# B&R Automation Studio project prac3
Automation Studio 4.5.2.102; technology packages: Acp10Arnc0 5.2.1

## Configuration Config1

CPU 4PP065.0571-P74, AutomationRuntime D4.52, Build 4.1.2, Vc V4.52.0, Safety 1.6

### Task classes (Cpu.sw)
```
Cyclic#1 (cycle 2000 us, tolerance 0 us):
  ncsdcctrl <- ncsdcctrl.prg
Cyclic#4:
  Program <- Program.prg
NcDataObjects: acp10etxen <- acp10etxen.dob, gAxis01a <- gAxis01obj.gAxis01a.dob, gAxis01i <- gAxis01obj.gAxis01i.dob, gAxis02a <- gAxis02obj.gAxis02a.dob, gAxis02i <- gAxis02obj.gAxis02i.dob, gAxis03a <- gAxis03obj.gAxis03a.dob, gAxis03i <- gAxis03obj.gAxis03i.dob, gAxis04a <- gAxis04obj.gAxis04a.dob, gAxis04i <- gAxis04obj.gAxis04i.dob
VcDataObjects: Visu <- Visu.dob
Libraries: Acp10man, Acp10par, NcGlobal, Acp10sdc, Acp10_MC, brsystem, sys_lib, runtime, AsBrStr, Library
```

### Hardware
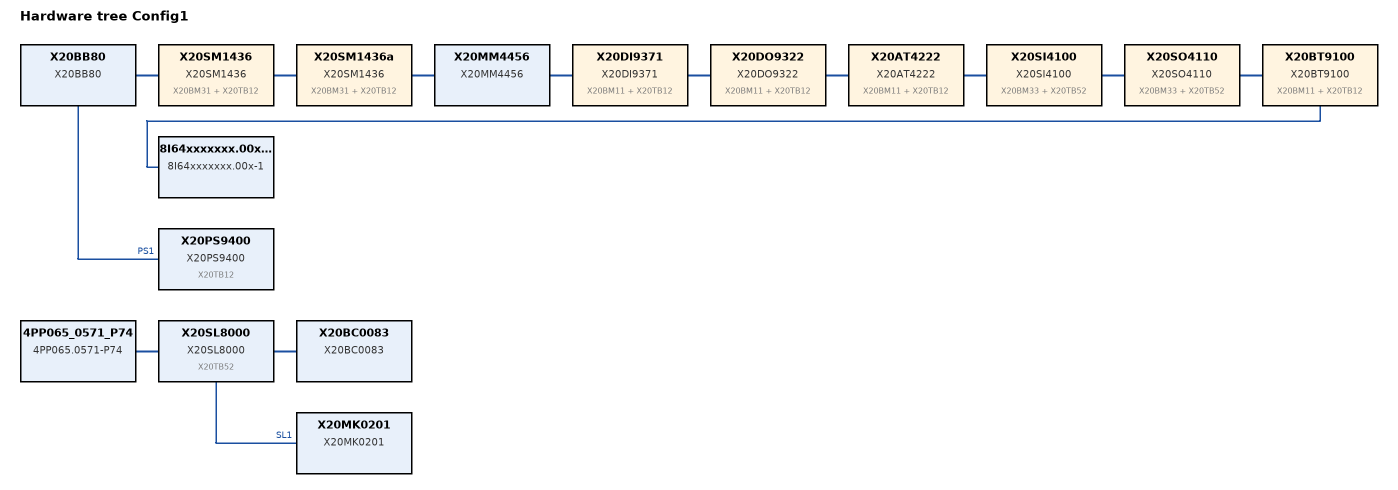
```
4PP065_0571_P74 : 4PP065.0571-P74 v1.1.2.0
  Connector IF5:
    ActivateDevice = 1
    Mode = Manual
    InternetAddress = 10.0.1.7
    SubnetMask = 255.255.255.0
  ConfigurationID = labBR
  TimerDeviceType = EPLX2X
  TimerDevice = 4PP065_0571_P74.IF4
  TaskClassIdleTime = 2000
  Cyclic1Duration = 2000
  Cyclic1Tolerance = 0
  Cyclic1Output = 1
  VcObjectName = Visu
8I64xxxxxxx.00x-1 : 8I64xxxxxxx.00x-1 v1.3.9.1  [X2X1 -> X20BT9100.X2X1 [Cable Type=X2XCable, Length=10, Version=1.0.0.2]]
  packedETAD = packed
  packedCMDD = packed
X20AT4222 : X20AT4222 v1.2.3.0  [SS1 -> X20TB12e.SS; SL -> X20BM11b.SL1]
X20BB80 : X20BB80 v1.0.2.0
X20BC0083 : X20BC0083 v2.9.0.0  [PLK1 -> X20SL8000.PLK2 [Cable Type=PowerlinkCable, Length=10, Version=1.0.0.2]; SL -> X20BB80.SL1]
X20BM11 : X20BM11 v1.0.0.1  [X2X1 -> X20MM4456.X2X2]
X20BM11a : X20BM11 v1.0.0.1  [X2X1 -> X20BM11.X2X2]
X20BM11b : X20BM11 v1.0.0.1  [X2X1 -> X20BM11a.X2X2]
X20BM11c : X20BM11 v1.0.0.1  [X2X1 -> X20BM33a.X2X2]
X20BM31 : X20BM31 v1.0.0.1  [X2X1 -> X20BB80.IF1]
X20BM31a : X20BM31 v1.0.0.1  [X2X1 -> X20BM31.X2X2]
X20BM33 : X20BM33 v1.0.0.4  [X2X1 -> X20BM11b.X2X2]
X20BM33a : X20BM33 v1.0.0.4  [X2X1 -> X20BM33.X2X2]
X20BT9100 : X20BT9100 v1.0.3.0  [SS1 -> X20TB12f.SS; SL -> X20BM11c.SL1]
X20DI9371 : X20DI9371 v1.0.2.0  [SS1 -> X20TB12c.SS; SL -> X20BM11.SL1]
X20DO9322 : X20DO9322 v1.0.3.0  [SS1 -> X20TB12d.SS; SL -> X20BM11a.SL1]
X20MK0201 : X20MK0201 v1.0.0.0  [SL -> X20SL8000.SL1]
X20MM4456 : X20MM4456 v1.4.0.0  [X2X1 -> X20BM31a.X2X2]
X20PS9400 : X20PS9400 v1.0.2.4  [SS1 -> X20TB12.SS; PS -> X20BB80.PS1]
X20SI4100 : X20SI4100 v1.10.1.1  [SS1 -> X20TB52a.SS; SL -> X20BM33.SL1]
X20SL8000 : X20SL8000 v1.6.5.1  [PLK1 -> 4PP065_0571_P74.IF4 [Cable Type=PowerlinkCable, Length=10, Version=1.0.0.2]; PLK2 -> X20BC0083.PLK1 [Cable Type=PowerlinkCable, Length=10, Version=1.0.0.2]; SS1 -> X20TB52.SS]
  SafeProject = SafeLOGIC-1
X20SM1436 : X20SM1436 v1.4.2.1  [SS1 -> X20TB12b.SS; SL -> X20BM31.SL1]
X20SM1436a : X20SM1436 v1.4.2.1  [SS1 -> X20TB12a.SS; SL -> X20BM31a.SL1]
X20SO4110 : X20SO4110 v1.10.1.1  [SS1 -> X20TB52b.SS; SL -> X20BM33a.SL1]
  SafeModuleID = 3
X20TB12 : X20TB12 v1.0.0.0
X20TB12a : X20TB12 v1.0.0.0
X20TB12b : X20TB12 v1.0.0.0
X20TB12c : X20TB12 v1.0.0.0
X20TB12d : X20TB12 v1.0.0.0
X20TB12e : X20TB12 v1.0.0.0
X20TB12f : X20TB12 v1.0.0.0
X20TB52 : X20TB52 v1.0.0.1
X20TB52a : X20TB52 v1.0.0.1
X20TB52b : X20TB52 v1.0.0.1
```

### IoMap.iom - 4PP065_0571_P74/IoMap.iom
```iecst
VAR_CONFIG
	Cyclic#1.gAxis01_DrvIf.iLifeCnt AT %IB."X20SM1436".LifeCnt;
	Cyclic#1.gAxis01_DrvIf.iDrvOK AT %IX."X20SM1436".DrvOk01;
	Cyclic#1.gAxis01_DrvIf.oBoostCurrent AT %QX."X20SM1436".BoostCurrent01;
	Cyclic#1.gAxis01_DrvIf.oStandStillCurrent AT %QX."X20SM1436".StandstillCurrent01;
	Cyclic#1.gAxis01_DrvIf.oSetTime AT %QW."X20SM1436".SetTime01;
	Cyclic#1.gAxis01_MotorStep0 AT %QW."X20SM1436".Motor1Step0;
	Cyclic#1.gAxis01_DiDoIf.iLifeCntDriveEnable AT %IB."X20SM1436".LifeCnt;
	Cyclic#1.gAxis01_DiDoIf.iLifeCntDriveReady AT %IB."X20SM1436".LifeCnt;
	Cyclic#1.gAxis01_DiDoIf.iDriveReady AT %IX."X20SM1436".DrvOk01;
	Cyclic#1.gAxis01_DiDoIf.oDriveEnable AT %QX."X20SM1436".DriveEnable01;
	Cyclic#1.gAxis01_EncIf1.iLifeCnt AT %IB."X20SM1436".LifeCnt;
	Cyclic#1.gAxis01_EncIf1.iEncOK AT %IX."X20SM1436".EncOk01;
	Cyclic#1.gAxis01_EncIf1.iActPos AT %IW."X20SM1436".ActPos01;
	Cyclic#1.gAxis01_EncIf1.iRefPulsePos AT %IW."X20SM1436".RefPulsePos01;
	Cyclic#1.gAxis01_EncIf1.iRefPulseCnt AT %IB."X20SM1436".RefPulseCnt01;
	Cyclic#1.gAxis01_EncIf1.iActTime AT %IW."X20SM1436".ActTime01;
	Cyclic#1.gAxis02_DrvIf.iLifeCnt AT %IB."X20SM1436a".LifeCnt;
	Cyclic#1.gAxis02_DrvIf.iDrvOK AT %IX."X20SM1436a".DrvOk01;
	Cyclic#1.gAxis02_DrvIf.oBoostCurrent AT %QX."X20SM1436a".BoostCurrent01;
	Cyclic#1.gAxis02_DrvIf.oStandStillCurrent AT %QX."X20SM1436a".StandstillCurrent01;
	Cyclic#1.gAxis02_DrvIf.oSetTime AT %QW."X20SM1436a".SetTime01;
	Cyclic#1.gAxis02_MotorStep0 AT %QW."X20SM1436a".Motor1Step0;
	Cyclic#1.gAxis02_DiDoIf.iLifeCntDriveEnable AT %IB."X20SM1436a".LifeCnt;
	Cyclic#1.gAxis02_DiDoIf.iLifeCntDriveReady AT %IB."X20SM1436a".LifeCnt;
	Cyclic#1.gAxis02_DiDoIf.iDriveReady AT %IX."X20SM1436a".DrvOk01;
	Cyclic#1.gAxis02_DiDoIf.oDriveEnable AT %QX."X20SM1436a".DriveEnable01;
	Cyclic#1.gAxis02_EncIf1.iLifeCnt AT %IB."X20SM1436a".LifeCnt;
	Cyclic#1.gAxis02_EncIf1.iEncOK AT %IX."X20SM1436a".EncOk01;
	Cyclic#1.gAxis02_EncIf1.iActPos AT %IW."X20SM1436a".ActPos01;
	Cyclic#1.gAxis02_EncIf1.iRefPulsePos AT %IW."X20SM1436a".RefPulsePos01;
	Cyclic#1.gAxis02_EncIf1.iRefPulseCnt AT %IB."X20SM1436a".RefPulseCnt01;
	Cyclic#1.gAxis02_EncIf1.iActTime AT %IW."X20SM1436a".ActTime01;
	Cyclic#1.gAxis04_DrvIf.iLifeCnt AT %IB."8I64xxxxxxx.00x-1".SDC_LifeCnt;
	Cyclic#1.gAxis04_DrvIf.iDrvOK AT %IX."8I64xxxxxxx.00x-1".ETAD_Input_Bool_02;
	Cyclic#1.gAxis04_DrvIf.oSetTime AT %QW."8I64xxxxxxx.00x-1".SDC_SetTime;
	Cyclic#1.::Program:speed AT %QW."8I64xxxxxxx.00x-1".LFRD_Output;
	Cyclic#1.gAxis04_DiDoIf.iLifeCntDriveReady AT %IB."8I64xxxxxxx.00x-1".SDC_LifeCnt;
	Cyclic#1.gAxis04_DiDoIf.iLifeCntDriveEnable AT %IB."8I64xxxxxxx.00x-1".SDC_LifeCnt;
	Cyclic#1.gAxis04_DiDoIf.oDriveEnable AT %QX."8I64xxxxxxx.00x-1".CMDD_Output_Bool_00;
	Cyclic#1.gAxis04_ModuleOk AT %QX."8I64xxxxxxx.00x-1".CMDD_Output_Bool_01;
	Cyclic#1.gAxis04_ModuleOk AT %QX."8I64xxxxxxx.00x-1".CMDD_Output_Bool_02;
	Cyclic#1.gAxis04_ModuleOk AT %IX."8I64xxxxxxx.00x-1".ModuleOk;
	Cyclic#1.gAxis04_DiDoIf.oDriveEnable AT %QX."8I64xxxxxxx.00x-1".CMDD_Output_Bool_03;
	Cyclic#1.gAxis04_DiDoIf.iDriveReady AT %IX."8I64xxxxxxx.00x-1".ETAD_Input_Bool_02;
	::Program:DRIVE.STATE AT %IW."8I64xxxxxxx.00x-1".ETAD_Input;
	::Program:DRIVE.COM AT %QW."8I64xxxxxxx.00x-1".CMDD_Output;
END_VAR
```

### Acp10map.ncm - 4PP065_0571_P74/Motion/Acp10map.ncm
```
NcMapping (NcSwId=Acp10)
  NcObject gAxis01 (ModuleId=X20SM1436, ModuleAddress=SDC_IF1.ST1, Type=ncAXIS, Channel=1, AcoposSimulation=Off, InitParameter=gAxis01i, AcoposParameter=gAxis01a, Disabled=FALSE, ModuleDisabled=FALSE)
  NcObject gAxis02 (ModuleId=X20SM1436a, ModuleAddress=SDC_IF1.ST2, Type=ncAXIS, Channel=1, AcoposSimulation=Off, InitParameter=gAxis02i, AcoposParameter=gAxis02a, Disabled=FALSE, ModuleDisabled=FALSE)
  NcObject gAxis04 (ModuleId=8I64xxxxxxx.00x-1, ModuleAddress=SDC_IF1.ST3, Type=ncAXIS, Channel=1, AcoposSimulation=Off, InitParameter=gAxis04i, AcoposParameter=gAxis04a, Disabled=FALSE, ModuleDisabled=FALSE)
```

## Logical view

Binary libraries used (declarations not repeated): operator, runtime, astime, AsIecCon, Acp10man, Acp10par, NcGlobal, Acp10sdc, Acp10_MC, brsystem, sys_lib, AsBrStr

### Global.var - Global variables
```iecst
VAR
	gAxis01 : ACP10AXIS_typ;
	gAxis01_HW : SdcHwCfg_typ := (0);
	gAxis01_DrvIf : SdcDrvIf16_typ := (0);
	gAxis01_EncIf1 : SdcEncIf16_typ := (0);
	gAxis01_DiDoIf : SdcDiDoIf_typ := (0);
	gAxis01_MotorStep0 : INT := (0);
	gAxis02 : ACP10AXIS_typ;
	gAxis02_HW : SdcHwCfg_typ := (0);
	gAxis02_DrvIf : SdcDrvIf16_typ := (0);
	gAxis02_EncIf1 : SdcEncIf16_typ := (0);
	gAxis02_DiDoIf : SdcDiDoIf_typ := (0);
	gAxis02_MotorStep0 : INT := (0);
	gAxis03 : ACP10AXIS_typ;
	gAxis03_HW : SdcHwCfg_typ := (0);
	gAxis03_DrvIf : SdcDrvIf16_typ := (0);
	gAxis03_DiDoIf : SdcDiDoIf_typ := (0);
	gAxis03_ModuleOk : BOOL := 0;
	gAxis04 : ACP10AXIS_typ;
	gAxis04_HW : SdcHwCfg_typ := (0);
	gAxis04_DrvIf : SdcDrvIf16_typ := (0);
	gAxis04_DiDoIf : SdcDiDoIf_typ := (0);
	gAxis04_ModuleOk : BOOL := 0;
	ENABLED : BOOL := FALSE;
END_VAR
```

### Package Logical/Libraries - Global libraries

### Library Logical/Libraries/Library (ANSIC)

#### Constants.var - Exported constants
```iecst
VAR CONSTANT
	CMD_SWITCHED_ON : UINT := 7;
	CMD_DISABLE_VOLTAGE1 : UINT := 0;
	CMD_ENABLED : UINT := 15;
	CMD_SHUTDOWN : UINT := 6;
	STATE_READY : UINT := 33;
	STATE_DISABLED : UINT := 64;
	STATE_SWITCHED_ON : UINT := 35;
END_VAR
```

#### Library.fun - Exported functions and function blocks
```iecst
{REDUND_OK} FUNCTION_BLOCK drive (*TODO: Add your comment here*) (*$GROUP=User,$CAT=User,$GROUPICON=User.png,$CATICON=User.png*)
	VAR_INPUT
		ENABLE : BOOL;
		STATE : UINT;
	END_VAR
	VAR_OUTPUT
		COM : UINT;
	END_VAR
END_FUNCTION_BLOCK
```

#### drive.c
```c
#include <bur/plctypes.h>
#ifdef __cplusplus
	extern "C"
	{
#endif
	#include "Library.h"
#ifdef __cplusplus
	};
#endif
/* TODO: Add your comment here */
void drive(struct drive* inst)
{
	UINT mask=inst->STATE & 0x6f;
	if(!inst->ENABLE){
		inst->COM = CMD_SHUTDOWN;
	}
	else{
		switch(mask)
		{
			case STATE_DISABLED:
				inst->COM=CMD_SHUTDOWN;
				break;
			case STATE_READY:
				inst->COM=CMD_ENABLED;
				break;
			case STATE_SWITCHED_ON:
				inst->COM=CMD_SWITCHED_ON;
				break;

		}
	}
}
```

### Program Logical/ncsdcctrl (IEC)

#### ncsdcctrl.var
```iecst
VAR
	gAxis01_oSetPosOld : INT := 0;
	gAxis02_oSetPosOld : INT := 0;
END_VAR
```

#### ncsdcctrlCyclic.st
```iecst
PROGRAM _CYCLIC

(* ### BEGIN gAxis01 ### *)

(* life counter emulation of digital inputs *)
      gAxis01_DiDoIf.iLifeCntReference := gAxis01_DiDoIf.iLifeCntReference + 1;
      gAxis01_DiDoIf.iLifeCntNegHwEnd  := gAxis01_DiDoIf.iLifeCntNegHwEnd  + 1;
      gAxis01_DiDoIf.iLifeCntPosHwEnd  := gAxis01_DiDoIf.iLifeCntPosHwEnd  + 1;

(* default function model of ACOPOSmicro: convert absolute steps to delta steps - overflow save delta calculation *)
      gAxis01_MotorStep0 := gAxis01_DrvIf.oSetPos - gAxis01_oSetPosOld;
      gAxis01_oSetPosOld := gAxis01_DrvIf.oSetPos;

(* ### END gAxis01 ### *)

(* ### BEGIN gAxis02 ### *)

(* life counter emulation of digital inputs *)
      gAxis02_DiDoIf.iLifeCntReference := gAxis02_DiDoIf.iLifeCntReference + 1;
      gAxis02_DiDoIf.iLifeCntNegHwEnd  := gAxis02_DiDoIf.iLifeCntNegHwEnd  + 1;
      gAxis02_DiDoIf.iLifeCntPosHwEnd  := gAxis02_DiDoIf.iLifeCntPosHwEnd  + 1;

(* default function model of ACOPOSmicro: convert absolute steps to delta steps - overflow save delta calculation *)
      gAxis02_MotorStep0 := gAxis02_DrvIf.oSetPos - gAxis02_oSetPosOld;
      gAxis02_oSetPosOld := gAxis02_DrvIf.oSetPos;

(* ### END gAxis02 ### *)

(* ### BEGIN gAxis03 ### *)

(* life counter emulation of digital inputs *)
        gAxis03_DiDoIf.iLifeCntReference := gAxis03_DiDoIf.iLifeCntReference + 1;
        gAxis03_DiDoIf.iLifeCntNegHwEnd  := gAxis03_DiDoIf.iLifeCntNegHwEnd  + 1;
        gAxis03_DiDoIf.iLifeCntPosHwEnd  := gAxis03_DiDoIf.iLifeCntPosHwEnd  + 1;

(* ### END gAxis03 ### *)

(* ### BEGIN gAxis04 ### *)

(* life counter emulation of digital inputs *)
        gAxis04_DiDoIf.iLifeCntReference := gAxis04_DiDoIf.iLifeCntReference + 1;
        gAxis04_DiDoIf.iLifeCntNegHwEnd  := gAxis04_DiDoIf.iLifeCntNegHwEnd  + 1;
        gAxis04_DiDoIf.iLifeCntPosHwEnd  := gAxis04_DiDoIf.iLifeCntPosHwEnd  + 1;

(* ### END gAxis04 ### *)

END_PROGRAM
```

#### ncsdcctrlInit.st
```iecst
PROGRAM _INIT

(* ### BEGIN gAxis01 ### *)

(* initialize general interfaces *)
      gAxis01.size := gAxis01.size;
      gAxis01_HW.DrvIf_Typ := ncSDC_DRVSM16;
      brsstrcpy( ADR(gAxis01_HW.DrvIf_Name[0]), ADR('gAxis01_DrvIf') );
      gAxis01_HW.DiDoIf_Typ := ncSDC_DIDO;
      brsstrcpy( ADR(gAxis01_HW.DiDoIf_Name[0]), ADR('gAxis01_DiDoIf') );
      gAxis01_HW.EncIf1_Typ := ncSDC_ENC16;
      brsstrcpy( ADR(gAxis01_HW.EncIf1_Name[0]), ADR('gAxis01_EncIf1') );
      gAxis01_EncIf1.iLifeCnt := gAxis01_EncIf1.iLifeCnt;

(* initialize old-value for delta step calculation *)
      gAxis01_oSetPosOld := gAxis01_DrvIf.oSetPos;

(* ### END gAxis01 ### *)

(* ### BEGIN gAxis02 ### *)

(* initialize general interfaces *)
      gAxis02.size := gAxis02.size;
      gAxis02_HW.DrvIf_Typ := ncSDC_DRVSM16;
      brsstrcpy( ADR(gAxis02_HW.DrvIf_Name[0]), ADR('gAxis02_DrvIf') );
      gAxis02_HW.DiDoIf_Typ := ncSDC_DIDO;
      brsstrcpy( ADR(gAxis02_HW.DiDoIf_Name[0]), ADR('gAxis02_DiDoIf') );
      gAxis02_HW.EncIf1_Typ := ncSDC_ENC16;
      brsstrcpy( ADR(gAxis02_HW.EncIf1_Name[0]), ADR('gAxis02_EncIf1') );
      gAxis02_EncIf1.iLifeCnt := gAxis02_EncIf1.iLifeCnt;

(* initialize old-value for delta step calculation *)
      gAxis02_oSetPosOld := gAxis02_DrvIf.oSetPos;

(* ### END gAxis02 ### *)

(* ### BEGIN gAxis03 ### *)

(* initialize variables *)
        gAxis03_HW.DrvIf_Typ := ncSDC_DRVSERVO16;
        brsstrcpy(ADR(gAxis03_HW.DrvIf_Name[0]), ADR('gAxis03_DrvIf'));
        gAxis03_HW.DiDoIf_Typ := ncSDC_DIDO;
        brsstrcpy(ADR(gAxis03_HW.DiDoIf_Name[0]), ADR('gAxis03_DiDoIf'));

(* force variable offset generation *)
        gAxis03.size                      := gAxis03.size;
        gAxis03_DrvIf.iLifeCnt            := gAxis03_DrvIf.iLifeCnt;
        gAxis03_DiDoIf.iLifeCntDriveReady := gAxis03_DiDoIf.iLifeCntDriveReady;
        gAxis03_ModuleOk                  := gAxis03_ModuleOk;

(* assign your hardware inputs here*)

(*      gAxis03_DiDoIf.iPosHwEnd  := gAxis03_DiDoIf.iPosHwEnd;
        gAxis03_DiDoIf.iNegHwEnd  := gAxis03_DiDoIf.iNegHwEnd;
        gAxis03_DiDoIf.iReference := gAxis03_DiDoIf.iReference;
 *)

(* ### END gAxis03 ### *)

(* ### BEGIN gAxis04 ### *)

(* initialize variables *)
        gAxis04_HW.DrvIf_Typ := ncSDC_DRVSERVO16;
        brsstrcpy(ADR(gAxis04_HW.DrvIf_Name[0]), ADR('gAxis04_DrvIf'));
        gAxis04_HW.DiDoIf_Typ := ncSDC_DIDO;
        brsstrcpy(ADR(gAxis04_HW.DiDoIf_Name[0]), ADR('gAxis04_DiDoIf'));

(* force variable offset generation *)
        gAxis04.size                      := gAxis04.size;
        gAxis04_DrvIf.iLifeCnt            := gAxis04_DrvIf.iLifeCnt;
        gAxis04_DiDoIf.iLifeCntDriveReady := gAxis04_DiDoIf.iLifeCntDriveReady;
        gAxis04_ModuleOk                  := gAxis04_ModuleOk;

(* assign your hardware inputs here*)

(*      gAxis04_DiDoIf.iPosHwEnd  := gAxis04_DiDoIf.iPosHwEnd;
        gAxis04_DiDoIf.iNegHwEnd  := gAxis04_DiDoIf.iNegHwEnd;
        gAxis04_DiDoIf.iReference := gAxis04_DiDoIf.iReference;
 *)

(* ### END gAxis04 ### *)

END_PROGRAM
```


- Data object Logical/gAxis02obj/gAxis02a (Apt) (no source held here)

- Data object Logical/gAxis02obj/gAxis02i (Ax) (no source held here)

- Data object Logical/gAxis03obj/gAxis03a (Apt) (no source held here)

- Data object Logical/gAxis03obj/gAxis03i (Ax) (no source held here)

- Data object Logical/gAxis04obj/gAxis04a (Apt) (no source held here)

- Data object Logical/gAxis04obj/gAxis04i (Ax) (no source held here)

### Program Logical/Program (ANSIC)

#### Variables.var
```iecst
VAR
	speed : INT;
	DRIVE : drive;
END_VAR
```

#### Main.c
```c
#include <bur/plctypes.h>

#ifdef _DEFAULT_INCLUDES
	#include <AsDefault.h>
#endif

void _INIT ProgramInit(void)
{
	speed=400;
	DRIVE.ENABLE=0;
}

void _CYCLIC ProgramCyclic(void)
{
	DRIVE.ENABLE = ENABLED;
	drive(&DRIVE);
}

void _EXIT ProgramExit(void)
{

}
```

- Visualisation Logical/Visu (not shown)

Listed in the project but not available here: Logical/Global.typ, Logical/Libraries/Library/Types.typ, Logical/acp10etxen, Logical/gAxis01obj
